// TIA Portal V17 export
// export: Created 2025-08-05T09:36:01.0298833Z, ExportSetting WithDefaults, DisplayName Totally Integrated Automation Portal, DisplayVersion V17, DisplayName TIA Portal Openness, DisplayVersion V17, DisplayName TIA Portal Version Control Interface, DisplayVersion V17, DisplayName SINAMICS Startdrive Advanced, DisplayVersion V17, DisplayName SINAMICS Startdrive G130, G150, S120, S150, SINAMICS MV, S210, DisplayVersion V17, DisplayName SINAMICS Startdrive G110M, G120, G120C, G120D, G120P, G115D, DisplayVersion V17, DisplayName STEP 7 Professional, DisplayVersion V17, DisplayName STEP 7 Safety, DisplayVersion V17, DisplayName WinCC Advanced, DisplayVersion V17
TYPE "typeMotion"
TITLE = Movement / Bewegung
// Movement [V 01.00 | Kernel_V2] / Bewegung [V 01.00 | Kernel_V2]
// stored: IsFailsafeCompliant false
   STRUCT
      autoToPos : Bool;   // Automatic to Position / Automatic to position
      inPosition : Bool;   // In Position / In position
      autoInPos : Bool;   // In Position Automatic / In position automatic
      toPosition : Bool;   // To Position
   END_STRUCT;
END_TYPE
